// Injects restored flags into an otherwise fresh instance. This exercises
// startup policy, not actual TwinCAT persistent-image durability.
FUNCTION_BLOCK FB_AlarmRestart_Probe EXTENDS TcForge.FB_AlarmSimple

SUPER^();

METHOD PUBLIC SeedSavedLatch
VAR_INPUT acknowledged : BOOL; END_VAR
_latchedSync := TRUE;
_ackedSync := acknowledged;
END_METHOD

END_FUNCTION_BLOCK

(* stored: Version 1.1.0.1
   POU FB_AlarmRestart_Probe: Id {13ed5234-aa7a-4314-b881-40fb364475e2}
   Method SeedSavedLatch: Id {488547cb-e058-44bd-ae2e-00f3ebd09ffb} *)
